# EPICS substitutions: ffmpegServer/iocs/ffmpegServerIOC/ffmpegServerApp/Db/example_expanded.substitutions
# This file was automatically generated on Thu 24 Jul 2014 16:29:02 BST from
# source: /home/up45/github/ffmpegServer/etc/makeIocs/example.xml
#
# *** Please do not edit this file: edit the source file instead. ***
#

# Macros:
#  P        Device Prefix
#  R        Device Suffix
#  PORT     Asyn Port name
#  TIMEOUT  Timeout
#  ADDR     Asyn Port address
file $(ADCORE)/db/ADBase.template
{
pattern { P, R, PORT, TIMEOUT, ADDR }
    { "BLxxI-DI-PHDGN-01", ":CAM:", "C1.CAM", "1", "0" }
}

# Macros:
#  P        Device Prefix
#  R        Device Suffix
#  PORT     Asyn Port name
#  TIMEOUT  Timeout
#  ADDR     Asyn Port address
file $(ADCORE)/db/simDetector.template
{
pattern { P, R, PORT, TIMEOUT, ADDR }
    { "BLxxI-DI-PHDGN-01", ":CAM:", "C1.CAM", "1", "0" }
}

# Macros:
#  P             Device Prefix
#  R             Device Suffix
#  PORT          Asyn Port name
#  TIMEOUT       Timeout
#  ADDR          Asyn Port address
#  NDARRAY_PORT  Input Array Port
#  NDARRAY_ADDR  Input Array Address
#  Enabled       Plugin Enabled at startup?
file $(ADCORE)/db/NDPluginBase.template
{
pattern { P, R, PORT, TIMEOUT, ADDR, NDARRAY_PORT, NDARRAY_ADDR, Enabled }
    { "BLxxI-DI-PHDGN-01", ":MJPG:", "C1.MJPG", "1", "0", "C1.CAM", "0", "1" }
    { "BLxxI-DI-PHDGN-01", ":FILE:", "C1.FILE", "1", "0", "C1.CAM", "0", "0" }
}

# Macros:
#  P        Device Prefix
#  R        Device Suffix
#  PORT     Asyn Port name
#  QUALITY  Jpeg Quality in percent
#  MAXW     Maximum Jpeg Width
#  MAXH     Maximum Jpeg Height
file $(FFMPEGSERVER)/db/ffmpegStream.template
{
pattern { P, R, PORT, QUALITY, MAXW, MAXH }
    { "BLxxI-DI-PHDGN-01", ":MJPG:", "C1.MJPG", "100", "1600", "1200" }
}

# Macros:
#  P        Device Prefix
#  R        Device Suffix
#  PORT     Asyn Port name
#  TIMEOUT  Timeout
#  ADDR     Asyn Port address
file $(ADCORE)/db/NDFile.template
{
pattern { P, R, PORT, TIMEOUT, ADDR }
    { "BLxxI-DI-PHDGN-01", ":FILE:", "C1.FILE", "1", "0" }
}

# Macros:
#  P     Device Prefix
#  R     Device Suffix
#  PORT  Asyn Port name
file $(FFMPEGSERVER)/db/ffmpegFile.template
{
pattern { P, R, PORT }
    { "BLxxI-DI-PHDGN-01", ":FILE:", "C1.FILE" }
}
